FUNCTION_BLOCK FB_Leitungswahl
VAR_INPUT
	I_Ventil_1		:FB_A_Magnetventil;
	I_Ventil_2		:FB_A_Magnetventil;
END_VAR
VAR_OUTPUT
	O_Ventil		:FB_A_Magnetventil;
END_VAR
VAR
END_VAR

IF P_Leitung = 1 THEN
	O_Ventil := I_Ventil_1;
ELSIF P_LEitung = 2 THEN
	O_Ventil := I_Ventil_2;
END_IF

PROPERTY P_Leitung : INT
SET
IF
END_SET
END_PROPERTY

END_FUNCTION_BLOCK

(* stored: Version 1.1.0.1, ProductVersion 3.1.4024.12
   POU FB_Leitungswahl: Id {a328e0e1-c3d6-4f17-a6f9-781f0fbe9cd7}, SpecialFunc None
   Property P_Leitung: Id {4ec915d3-da03-4ec6-86d9-808616c9712f}
   Set Set: Id {662614df-37de-4f73-8568-012e967d1118} *)
